TYPE Barcode_Station_DUT :
STRUCT
	Start:	BOOL;
	Ready:	BOOL;
	Running:	BOOL;
	Done:	BOOL;
	Valid:	BOOL;
	Reading_Gate_number:	STRING;
	Reading_Gate_number_OLD:	STRING;
	Number_OF_Reading_Gates:	STRING;
	Number_OF_Reading_Gates_OLD:	STRING;
	Barcode:	STRING;
	Barcode_Old:	STRING;
END_STRUCT
END_TYPE

(* stored: Version 1.1.0.1
   DUT Barcode_Station_DUT: Id {402cf4f0-ec72-4303-95a1-765419dd60ec} *)
